{attribute 'GeneratedUsingTerminal: CX1100-0004-0000'}
{attribute addProperty BoxType "CX1100-0004-0000"}
{attribute addProperty Id "EtcSlaveTerminalBaseInfoDataAT %I*InfoData_6F19DB2B2"}
{attribute addProperty CRC "2874840167"}
{attribute addProperty Size "2"}
TYPE CX1100_AB5A9467 EXTENDS EtcSlaveTerminalBase :
STRUCT
	{attribute addProperty Name "InfoData"}
	InfoData : InfoData_6F19DB2B;
END_STRUCT
END_TYPE

(* stored: Version 1.2.0.0, ProductVersion 3.1.4024.9
   DUT CX1100_AB5A9467: Id {16900661-9307-4a22-aab7-f237f644aebe} *)
